{attribute 'GeneratedUsingTerminal: EPP1332-0001-0017'}
{attribute addProperty BoxType "EPP1332-0001-0017"}
{attribute addProperty Id "A_0023_EPP1342_0001_0016A_0023_EPP1342_0001_0016_655E23A6322"}
{attribute addProperty CRC "3107792638"}
{attribute addProperty Size "322"}
TYPE A_0022_EPP1332_0001_0017_B93D26FE EXTENDS EPP1332_1FC0878B :
STRUCT
	{attribute addProperty Name "A_0023_EPP1342_0001_0016"}
	{attribute addProperty PreviousPort "A_0022(EPP1332-0001-0017) : D"}
	A_0023_EPP1342_0001_0016 : A_0023_EPP1342_0001_0016_655E23A6;
END_STRUCT
END_TYPE

(* stored: Version 1.2.0.0, ProductVersion 3.1.4024.9
   DUT A_0022_EPP1332_0001_0017_B93D26FE: Id {47edac31-ff56-4d32-b4fa-3d8043b1b916} *)
